SYSTEM DRILL_MVCDR (* Drill System Control+Diagnostics+HMI with Remote Model+View *)
  (* Standard: 61499-1; Classification: Simulation; ApplicationDomain: Transfer Lines; Function: Drilling *)
  (* Version 0.1, 2004-10-19, JHC, Rockwell Automation, Extended from DRILL_MVCDL. *)
  (* Version 0.0, 2004-09-28, JHC, Rockwell Automation, Extended from DRILL_MVCDL1. *)
  DEVICE MODEL : RMT_FRAME
    RESOURCE CLOCK : EMB_RES
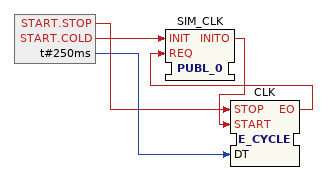
      FBS
        CLK : E_CYCLE;
        SIM_CLK : PUBL_0;
      END_FBS
      EVENT_CONNECTIONS
        START.STOP TO CLK.STOP;
        START.COLD TO SIM_CLK.INIT;
        SIM_CLK.INITO TO CLK.START;
        CLK.EO TO SIM_CLK.REQ;
      END_CONNECTIONS
      DATA_CONNECTIONS
        t#250ms TO CLK.DT;
      END_CONNECTIONS
    END_RESOURCE
    RESOURCE SENSORS : EMB_RES (* Sensor Data Concentrator/Publisher *)
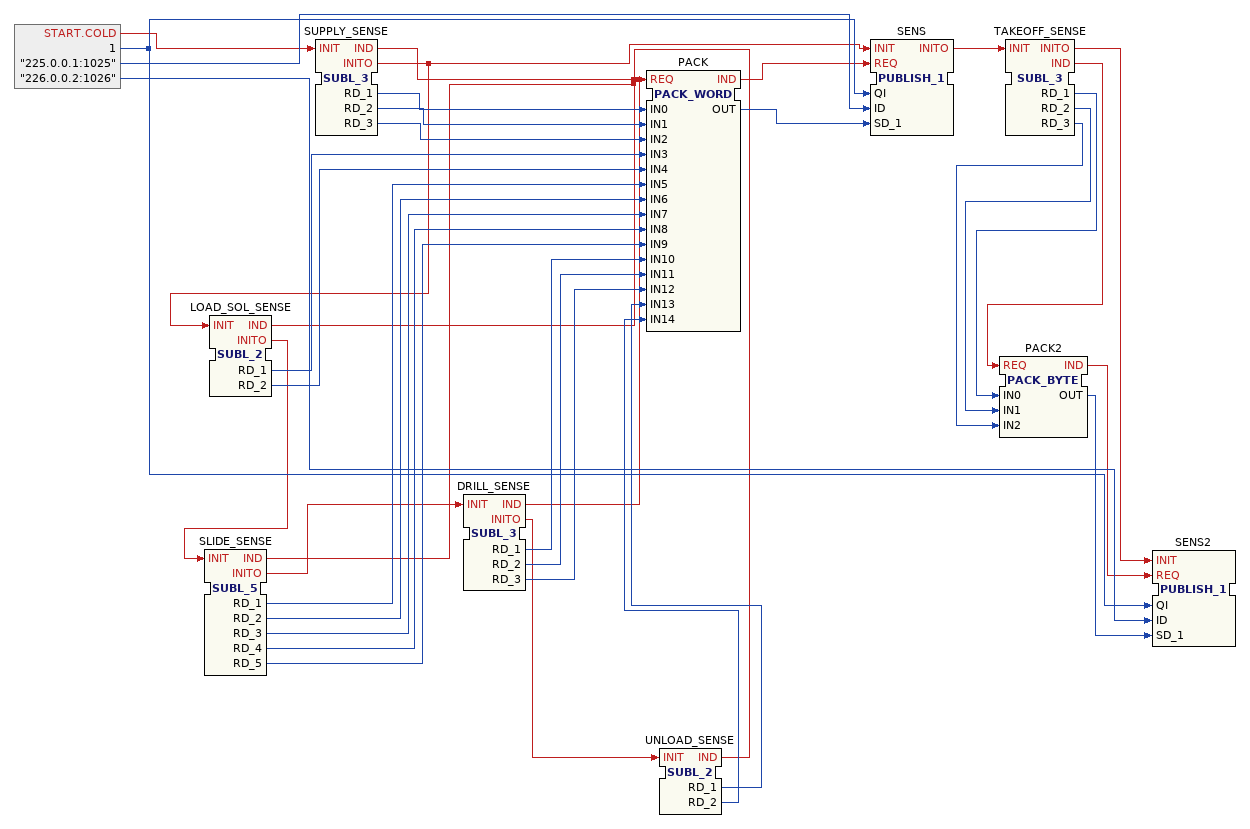
      FBS
        PACK : PACK_WORD;
        SENS : PUBLISH_1;
        SUPPLY_SENSE : SUBL_3;
        LOAD_SOL_SENSE : SUBL_2;
        SLIDE_SENSE : SUBL_5;
        DRILL_SENSE : SUBL_3;
        UNLOAD_SENSE : SUBL_2;
        SENS2 : PUBLISH_1;
        PACK2 : PACK_BYTE;
        TAKEOFF_SENSE : SUBL_3;
      END_FBS
      EVENT_CONNECTIONS
        SUPPLY_SENSE.IND TO PACK.REQ;
        LOAD_SOL_SENSE.IND TO PACK.REQ;
        SLIDE_SENSE.IND TO PACK.REQ;
        START.COLD TO SUPPLY_SENSE.INIT;
        DRILL_SENSE.IND TO PACK.REQ;
        SUPPLY_SENSE.INITO TO LOAD_SOL_SENSE.INIT;
        LOAD_SOL_SENSE.INITO TO SLIDE_SENSE.INIT;
        SLIDE_SENSE.INITO TO DRILL_SENSE.INIT;
        DRILL_SENSE.INITO TO UNLOAD_SENSE.INIT;
        UNLOAD_SENSE.IND TO PACK.REQ;
        SUPPLY_SENSE.INITO TO SENS.INIT;
        SENS.INITO TO TAKEOFF_SENSE.INIT;
        TAKEOFF_SENSE.INITO TO SENS2.INIT;
        PACK.IND TO SENS.REQ;
        TAKEOFF_SENSE.IND TO PACK2.REQ;
        PACK2.IND TO SENS2.REQ;
      END_CONNECTIONS
      DATA_CONNECTIONS
        SUPPLY_SENSE.RD_1 TO PACK.IN0;
        SUPPLY_SENSE.RD_2 TO PACK.IN1;
        SUPPLY_SENSE.RD_3 TO PACK.IN2;
        LOAD_SOL_SENSE.RD_1 TO PACK.IN3;
        LOAD_SOL_SENSE.RD_2 TO PACK.IN4;
        SLIDE_SENSE.RD_1 TO PACK.IN5;
        SLIDE_SENSE.RD_2 TO PACK.IN6;
        SLIDE_SENSE.RD_3 TO PACK.IN7;
        SLIDE_SENSE.RD_4 TO PACK.IN8;
        SLIDE_SENSE.RD_5 TO PACK.IN9;
        DRILL_SENSE.RD_1 TO PACK.IN10;
        DRILL_SENSE.RD_2 TO PACK.IN11;
        DRILL_SENSE.RD_3 TO PACK.IN12;
        UNLOAD_SENSE.RD_1 TO PACK.IN13;
        UNLOAD_SENSE.RD_2 TO PACK.IN14;
        1 TO SENS.QI;
        "225.0.0.1:1025" TO SENS.ID;
        PACK.OUT TO SENS.SD_1;
        TAKEOFF_SENSE.RD_1 TO PACK2.IN0;
        TAKEOFF_SENSE.RD_2 TO PACK2.IN1;
        TAKEOFF_SENSE.RD_3 TO PACK2.IN2;
        1 TO SENS2.QI;
        "226.0.0.2:1026" TO SENS2.ID;
        PACK2.OUT TO SENS2.SD_1;
      END_CONNECTIONS
    END_RESOURCE
    RESOURCE ACTUATORS : EMB_RES (* Actuator Data Subscriber/Distributor *)
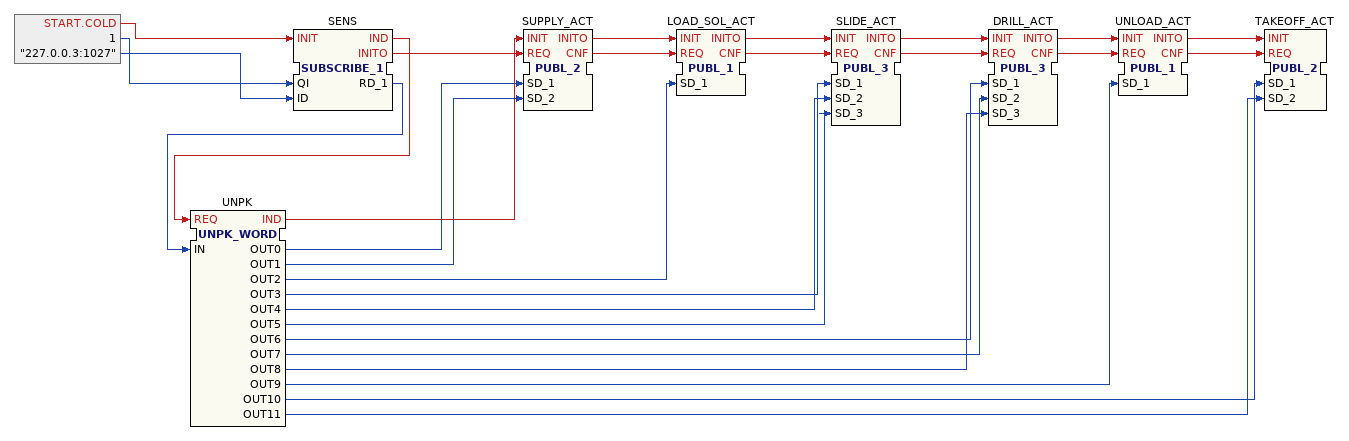
      FBS
        UNPK : UNPK_WORD;
        SENS : SUBSCRIBE_1;
        SUPPLY_ACT : PUBL_2;
        LOAD_SOL_ACT : PUBL_1;
        SLIDE_ACT : PUBL_3;
        DRILL_ACT : PUBL_3;
        UNLOAD_ACT : PUBL_1;
        TAKEOFF_ACT : PUBL_2;
      END_FBS
      EVENT_CONNECTIONS
        START.COLD TO SENS.INIT;
        SENS.IND TO UNPK.REQ;
        SENS.INITO TO SUPPLY_ACT.INIT;
        UNPK.IND TO SUPPLY_ACT.REQ;
        SUPPLY_ACT.INITO TO LOAD_SOL_ACT.INIT;
        SUPPLY_ACT.CNF TO LOAD_SOL_ACT.REQ;
        LOAD_SOL_ACT.INITO TO SLIDE_ACT.INIT;
        LOAD_SOL_ACT.CNF TO SLIDE_ACT.REQ;
        SLIDE_ACT.INITO TO DRILL_ACT.INIT;
        SLIDE_ACT.CNF TO DRILL_ACT.REQ;
        DRILL_ACT.INITO TO UNLOAD_ACT.INIT;
        DRILL_ACT.CNF TO UNLOAD_ACT.REQ;
        UNLOAD_ACT.INITO TO TAKEOFF_ACT.INIT;
        UNLOAD_ACT.CNF TO TAKEOFF_ACT.REQ;
      END_CONNECTIONS
      DATA_CONNECTIONS
        1 TO SENS.QI;
        "227.0.0.3:1027" TO SENS.ID;
        SENS.RD_1 TO UNPK.IN;
        UNPK.OUT0 TO SUPPLY_ACT.SD_1;
        UNPK.OUT1 TO SUPPLY_ACT.SD_2;
        UNPK.OUT2 TO LOAD_SOL_ACT.SD_1;
        UNPK.OUT3 TO SLIDE_ACT.SD_1;
        UNPK.OUT4 TO SLIDE_ACT.SD_2;
        UNPK.OUT5 TO SLIDE_ACT.SD_3;
        UNPK.OUT6 TO DRILL_ACT.SD_1;
        UNPK.OUT7 TO DRILL_ACT.SD_2;
        UNPK.OUT8 TO DRILL_ACT.SD_3;
        UNPK.OUT9 TO UNLOAD_ACT.SD_1;
        UNPK.OUT10 TO TAKEOFF_ACT.SD_1;
        UNPK.OUT11 TO TAKEOFF_ACT.SD_2;
      END_CONNECTIONS
    END_RESOURCE
    RESOURCE SUPPLY_MDL : EMB_RES
      FBS
        SUPPLY : XBAR_MDLL;
        LOAD_SOL : SOL_MDLL;
        UNLD : E_R_TRIG;
        LOAD : E_R_TRIG;
        SUPPLY_LOAD : LOADL;
      END_FBS
      EVENT_CONNECTIONS
        START.COLD TO SUPPLY.INIT;
        LOAD_SOL.IND TO UNLD.EI;
        SUPPLY.IND TO LOAD.EI;
        UNLD.EO TO SUPPLY.UNLD;
        SUPPLY.INITO TO SUPPLY_LOAD.INIT;
        SUPPLY_LOAD.INITO TO LOAD_SOL.INIT;
        LOAD_SOL.INITO TO SUPPLY_LOAD.REQ;
        LOAD.EO TO SUPPLY_LOAD.REQ;
      END_CONNECTIONS
      DATA_CONNECTIONS
        34 TO LOAD_SOL.VF;
        50 TO LOAD_SOL.VR;
        LOAD_SOL.END TO UNLD.QI;
        5 TO SUPPLY.VF;
        10 TO SUPPLY.VR;
        SUPPLY.HOME TO LOAD.QI;
        0 TO SUPPLY_LOAD.LPOS;
        VSTYLE#DISC TO SUPPLY_LOAD.STYLE;
        [255,255,0] TO SUPPLY_LOAD.WKPC;
      END_CONNECTIONS
    END_RESOURCE
    RESOURCE SLIDE_MDL : EMB_RES
      FBS
        SLIDE : XSLIDE_MDLL;
        UNLOAD : SOL_MDLL;
        DRILL_SENSE : SUBL_3;
        MAKE_HOLE : E_R_TRIG;
        UNLD : E_R_TRIG;
        LOAD_SOL_SENSE : SUBL_2;
        LOAD : E_R_TRIG;
        SLIDE_LOAD : LOADL;
        DRILLIT : LOADL;
      END_FBS
      EVENT_CONNECTIONS
        DRILL_SENSE.IND TO MAKE_HOLE.EI;
        UNLOAD.IND TO UNLD.EI;
        UNLD.EO TO SLIDE.UNLD;
        LOAD_SOL_SENSE.IND TO LOAD.EI;
        START.COLD TO UNLOAD.INIT;
        UNLOAD.INITO TO SLIDE.INIT;
        SLIDE.INITO TO LOAD_SOL_SENSE.INIT;
        LOAD_SOL_SENSE.INITO TO SLIDE_LOAD.INIT;
        LOAD.EO TO SLIDE_LOAD.REQ;
        MAKE_HOLE.EO TO DRILLIT.REQ;
        DRILLIT.INITO TO SLIDE.UNLD;
        SLIDE_LOAD.INITO TO DRILL_SENSE.INIT;
        DRILL_SENSE.INITO TO DRILLIT.INIT;
      END_CONNECTIONS
      DATA_CONNECTIONS
        50 TO UNLOAD.VF;
        50 TO UNLOAD.VR;
        DRILL_SENSE.RD_2 TO MAKE_HOLE.QI;
        20 TO SLIDE.VF;
        20 TO SLIDE.VR;
        UNLOAD.END TO UNLD.QI;
        LOAD_SOL_SENSE.RD_2 TO LOAD.QI;
        0 TO SLIDE_LOAD.LPOS;
        VSTYLE#DISC TO SLIDE_LOAD.STYLE;
        [255,255,0] TO SLIDE_LOAD.WKPC;
        "SLIDE_LOAD" TO DRILLIT.ID;
        100 TO DRILLIT.LPOS;
        VSTYLE#RING TO DRILLIT.STYLE;
        [255,255,0] TO DRILLIT.WKPC;
      END_CONNECTIONS
    END_RESOURCE
    RESOURCE DRILL_MDL : EMB_RES
      FBS
        DRILL : XBAR_MDLL;
        DRILL_ACT : SUBL_3;
        TOOL : E_SWITCH;
        DRILL_LOAD : LOADL;
        DRILL_UNLD : LOADL;
      END_FBS
      EVENT_CONNECTIONS
        START.COLD TO DRILL_ACT.INIT;
        DRILL_ACT.INITO TO DRILL.INIT;
        DRILL.INITO TO DRILL_LOAD.INIT;
        DRILL_LOAD.INITO TO DRILL_UNLD.INIT;
        DRILL_ACT.IND TO TOOL.EI;
        TOOL.EO1 TO DRILL_LOAD.REQ;
        TOOL.EO0 TO DRILL_UNLD.REQ;
        DRILL_UNLD.INITO TO DRILL_UNLD.REQ;
      END_CONNECTIONS
      DATA_CONNECTIONS
        10 TO DRILL.VF;
        15 TO DRILL.VR;
        VSTYLE#TOOL_ON TO DRILL_LOAD.STYLE;
        [255,255,0] TO DRILL_LOAD.WKPC;
        "DRILL_LOAD" TO DRILL_UNLD.ID;
        VSTYLE#TOOL_OFF TO DRILL_UNLD.STYLE;
        [255,255,0] TO DRILL_UNLD.WKPC;
        DRILL_ACT.RD_3 TO TOOL.G;
      END_CONNECTIONS
    END_RESOURCE
    RESOURCE TAKEOFF_MDL : EMB_RES
      FBS
        UNLOAD_SENSE : SUBL_2;
        TAKEOFF : XBAR_MDLL;
        UNLD : E_R_TRIG;
        LOAD : E_R_TRIG;
        TAKEOFF_LOAD : LOADL;
      END_FBS
      EVENT_CONNECTIONS
        START.COLD TO UNLOAD_SENSE.INIT;
        UNLD.EO TO TAKEOFF.UNLD;
        TAKEOFF.IND TO UNLD.EI;
        TAKEOFF.INITO TO TAKEOFF.UNLD;
        UNLOAD_SENSE.IND TO LOAD.EI;
        UNLOAD_SENSE.INITO TO TAKEOFF_LOAD.INIT;
        TAKEOFF_LOAD.INITO TO TAKEOFF.INIT;
        LOAD.EO TO TAKEOFF_LOAD.REQ;
      END_CONNECTIONS
      DATA_CONNECTIONS
        TAKEOFF.END TO UNLD.QI;
        10 TO TAKEOFF.VF;
        10 TO TAKEOFF.VR;
        UNLOAD_SENSE.RD_2 TO LOAD.QI;
        0 TO TAKEOFF_LOAD.LPOS;
        VSTYLE#RING TO TAKEOFF_LOAD.STYLE;
        [255,255,0] TO TAKEOFF_LOAD.WKPC;
      END_CONNECTIONS
    END_RESOURCE
    RESOURCE INPUT_VIEW : VIEW_PANEL
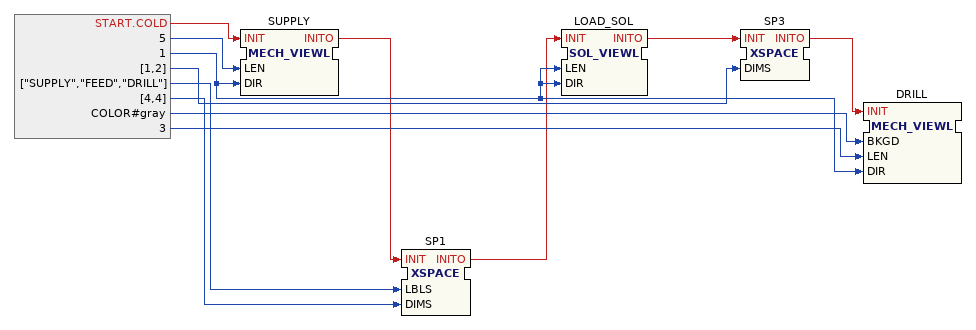
      FBS
        SUPPLY : MECH_VIEWL; (* Supply transfer mechanism *)
        SP1 : XSPACE;
        LOAD_SOL : SOL_VIEWL; (* Loader mechanism *)
        SP3 : XSPACE;
        DRILL : MECH_VIEWL;
      END_FBS
      EVENT_CONNECTIONS
        START.COLD TO SUPPLY.INIT;
        SUPPLY.INITO TO SP1.INIT;
        SP1.INITO TO LOAD_SOL.INIT;
        LOAD_SOL.INITO TO SP3.INIT;
        SP3.INITO TO DRILL.INIT;
      END_CONNECTIONS
      DATA_CONNECTIONS
        5 TO SUPPLY.LEN;
        1 TO SUPPLY.DIR;
        [1,2] TO SP3.DIMS;
        ["SUPPLY","FEED","DRILL"] TO SP1.LBLS;
        [4,4] TO SP1.DIMS;
        COLOR#gray TO DRILL.BKGD;
        3 TO DRILL.LEN;
        1 TO DRILL.DIR;
        1 TO LOAD_SOL.LEN;
        1 TO LOAD_SOL.DIR;
      END_CONNECTIONS
    END_RESOURCE
    RESOURCE OUTPUT_VIEW : VIEW_PANEL
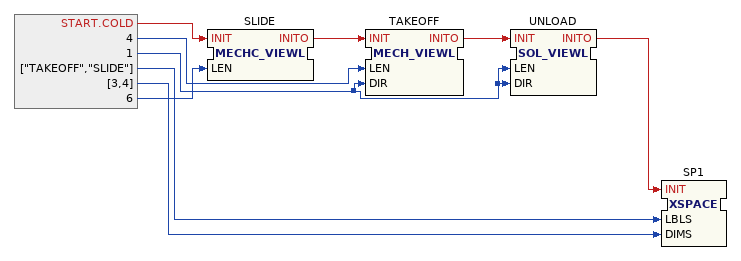
      FBS
        SLIDE : MECHC_VIEWL;
        TAKEOFF : MECH_VIEWL; (* Takeoff Transfer *)
        UNLOAD : SOL_VIEWL; (* Unloader Mechanism *)
        SP1 : XSPACE;
      END_FBS
      EVENT_CONNECTIONS
        START.COLD TO SLIDE.INIT;
        SLIDE.INITO TO TAKEOFF.INIT;
        TAKEOFF.INITO TO UNLOAD.INIT;
        UNLOAD.INITO TO SP1.INIT;
      END_CONNECTIONS
      DATA_CONNECTIONS
        4 TO TAKEOFF.LEN;
        1 TO TAKEOFF.DIR;
        ["TAKEOFF","SLIDE"] TO SP1.LBLS;
        [3,4] TO SP1.DIMS;
        1 TO UNLOAD.LEN;
        1 TO UNLOAD.DIR;
        6 TO SLIDE.LEN;
      END_CONNECTIONS
    END_RESOURCE
    DATA_CONNECTIONS
      0 TO INPUT_VIEW.TRACE;
      30 TO INPUT_VIEW.DIA;
      [6,5] TO INPUT_VIEW.SIZE;
      1 TO INPUT_VIEW.VERTICAL;
      30 TO OUTPUT_VIEW.DIA;
      [6,5] TO OUTPUT_VIEW.SIZE;
    END_CONNECTIONS
  END_DEVICE
  DEVICE DIAGNOSTICS : FRAME_DEVICE
    RESOURCE LOG : PANEL_RESOURCE
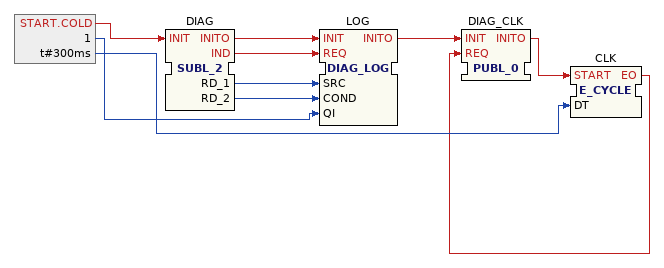
      FBS
        DIAG : SUBL_2;
        LOG : DIAG_LOG;
        CLK : E_CYCLE;
        DIAG_CLK : PUBL_0;
      END_FBS
      EVENT_CONNECTIONS
        START.COLD TO DIAG.INIT;
        DIAG.INITO TO LOG.INIT;
        DIAG.IND TO LOG.REQ;
        LOG.INITO TO DIAG_CLK.INIT;
        DIAG_CLK.INITO TO CLK.START;
        CLK.EO TO DIAG_CLK.REQ;
      END_CONNECTIONS
      DATA_CONNECTIONS
        DIAG.RD_1 TO LOG.SRC;
        DIAG.RD_2 TO LOG.COND;
        1 TO LOG.QI;
        t#300ms TO CLK.DT; (* Stretched 20% from MODEL.CLOCK.CLK.DT *)
      END_CONNECTIONS
    END_RESOURCE
    RESOURCE MONITOR : EMB_RES
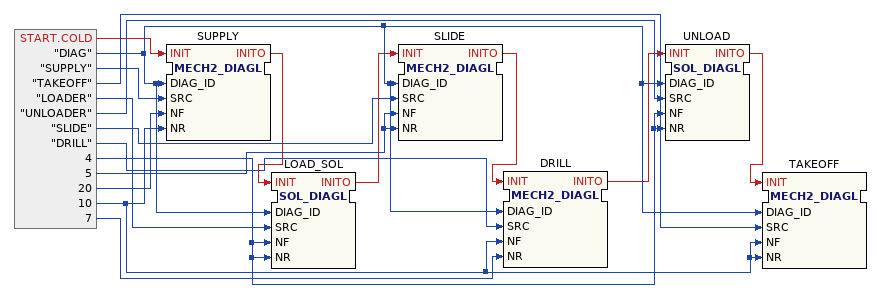
      FBS
        SUPPLY : MECH2_DIAGL;
        LOAD_SOL : SOL_DIAGL;
        SLIDE : MECH2_DIAGL;
        DRILL : MECH2_DIAGL;
        UNLOAD : SOL_DIAGL;
        TAKEOFF : MECH2_DIAGL;
      END_FBS
      EVENT_CONNECTIONS
        START.COLD TO SUPPLY.INIT;
        SUPPLY.INITO TO LOAD_SOL.INIT;
        LOAD_SOL.INITO TO SLIDE.INIT;
        SLIDE.INITO TO DRILL.INIT;
        DRILL.INITO TO UNLOAD.INIT;
        UNLOAD.INITO TO TAKEOFF.INIT;
      END_CONNECTIONS
      DATA_CONNECTIONS
        "DIAG" TO SUPPLY.DIAG_ID;
        "SUPPLY" TO SUPPLY.SRC;
        "DIAG" TO TAKEOFF.DIAG_ID;
        "TAKEOFF" TO TAKEOFF.SRC;
        "DIAG" TO LOAD_SOL.DIAG_ID;
        "LOADER" TO LOAD_SOL.SRC;
        "DIAG" TO UNLOAD.DIAG_ID;
        "UNLOADER" TO UNLOAD.SRC;
        "DIAG" TO SLIDE.DIAG_ID;
        "SLIDE" TO SLIDE.SRC;
        "DIAG" TO DRILL.DIAG_ID;
        "DRILL" TO DRILL.SRC;
        4 TO UNLOAD.NF;
        4 TO UNLOAD.NR;
        4 TO LOAD_SOL.NF;
        4 TO LOAD_SOL.NR;
        5 TO SLIDE.NF;
        5 TO SLIDE.NR;
        20 TO SUPPLY.NF;
        10 TO SUPPLY.NR;
        10 TO TAKEOFF.NF;
        10 TO TAKEOFF.NR;
        10 TO DRILL.NF;
        7 TO DRILL.NR;
      END_CONNECTIONS
    END_RESOURCE
    RESOURCE CLAMP : EMB_RES (* Special Monitoring for Clamp *)
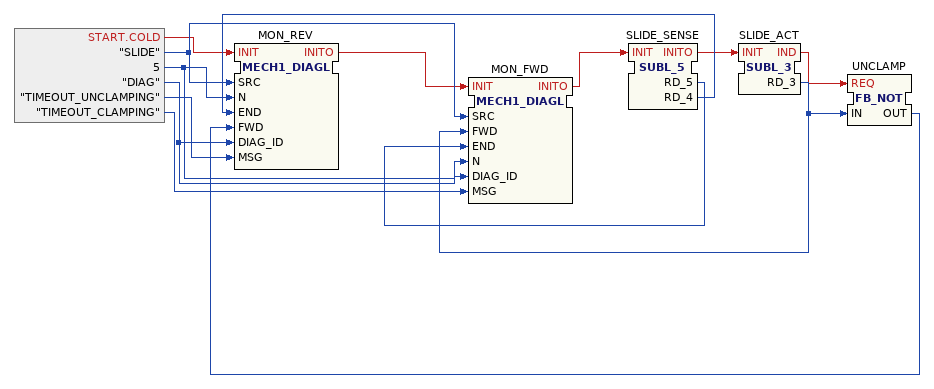
      FBS
        MON_FWD : MECH1_DIAGL;
        SLIDE_ACT : SUBL_3;
        SLIDE_SENSE : SUBL_5;
        MON_REV : MECH1_DIAGL;
        UNCLAMP : FB_NOT;
      END_FBS
      EVENT_CONNECTIONS
        SLIDE_ACT.IND TO UNCLAMP.REQ;
        SLIDE_SENSE.INITO TO SLIDE_ACT.INIT;
        START.COLD TO MON_REV.INIT;
        MON_REV.INITO TO MON_FWD.INIT;
        MON_FWD.INITO TO SLIDE_SENSE.INIT;
      END_CONNECTIONS
      DATA_CONNECTIONS
        "SLIDE" TO MON_FWD.SRC;
        "SLIDE" TO MON_REV.SRC;
        SLIDE_ACT.RD_3 TO UNCLAMP.IN;
        SLIDE_ACT.RD_3 TO MON_FWD.FWD;
        SLIDE_SENSE.RD_5 TO MON_FWD.END;
        5 TO MON_FWD.N;
        5 TO MON_REV.N;
        SLIDE_SENSE.RD_4 TO MON_REV.END;
        UNCLAMP.OUT TO MON_REV.FWD;
        "DIAG" TO MON_FWD.DIAG_ID;
        "DIAG" TO MON_REV.DIAG_ID;
        "TIMEOUT_UNCLAMPING" TO MON_REV.MSG;
        "TIMEOUT_CLAMPING" TO MON_FWD.MSG;
      END_CONNECTIONS
    END_RESOURCE
    RESOURCE SENSORS : EMB_RES (* Subscriber/Distributor for Sensors *)
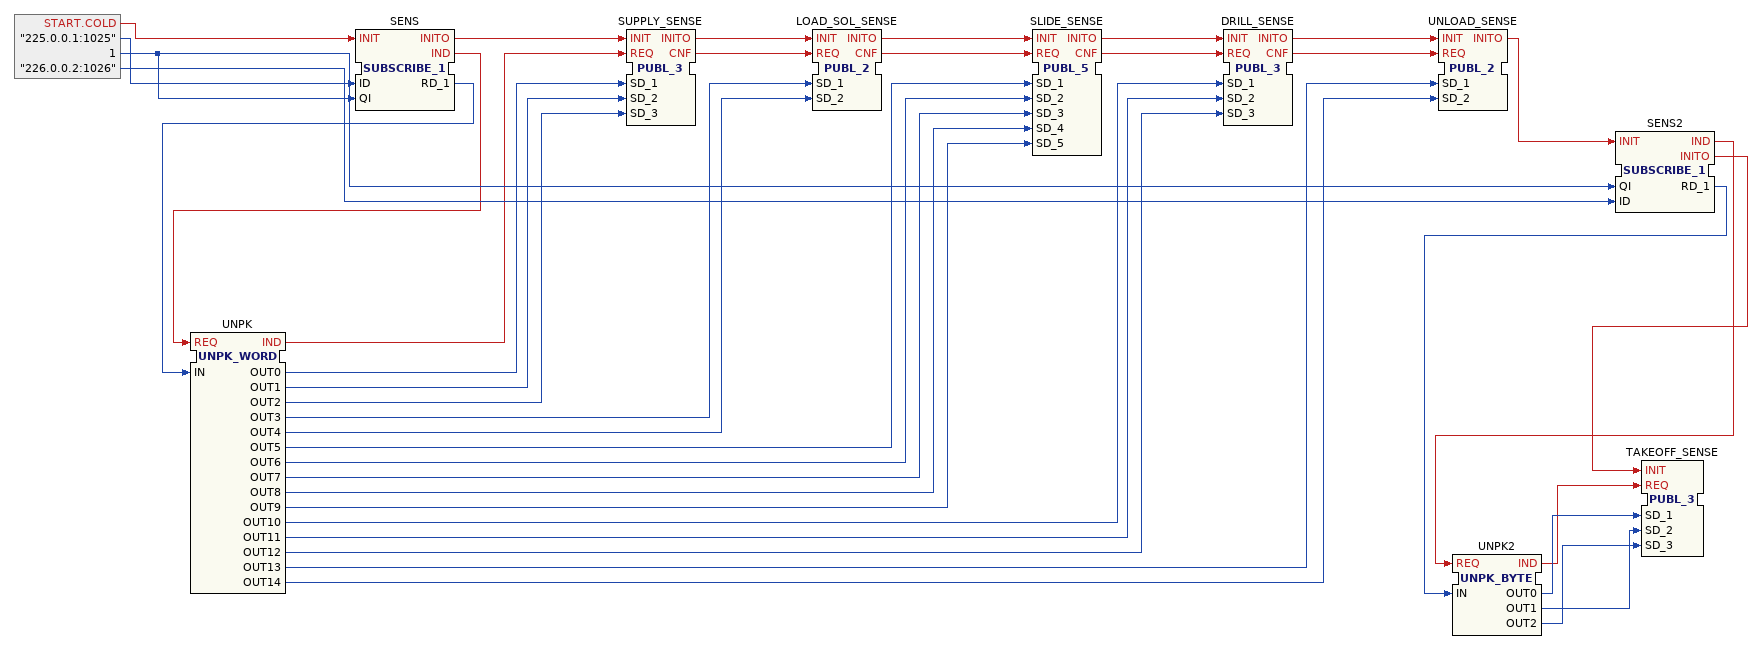
      FBS
        UNPK : UNPK_WORD;
        SENS : SUBSCRIBE_1;
        SUPPLY_SENSE : PUBL_3;
        LOAD_SOL_SENSE : PUBL_2;
        SLIDE_SENSE : PUBL_5;
        DRILL_SENSE : PUBL_3;
        UNLOAD_SENSE : PUBL_2;
        SENS2 : SUBSCRIBE_1;
        UNPK2 : UNPK_BYTE;
        TAKEOFF_SENSE : PUBL_3;
      END_FBS
      EVENT_CONNECTIONS
        START.COLD TO SENS.INIT;
        SENS.INITO TO SUPPLY_SENSE.INIT;
        SENS.IND TO UNPK.REQ;
        UNPK.IND TO SUPPLY_SENSE.REQ;
        SUPPLY_SENSE.INITO TO LOAD_SOL_SENSE.INIT;
        SUPPLY_SENSE.CNF TO LOAD_SOL_SENSE.REQ;
        LOAD_SOL_SENSE.INITO TO SLIDE_SENSE.INIT;
        LOAD_SOL_SENSE.CNF TO SLIDE_SENSE.REQ;
        SLIDE_SENSE.INITO TO DRILL_SENSE.INIT;
        SLIDE_SENSE.CNF TO DRILL_SENSE.REQ;
        DRILL_SENSE.INITO TO UNLOAD_SENSE.INIT;
        DRILL_SENSE.CNF TO UNLOAD_SENSE.REQ;
        UNLOAD_SENSE.INITO TO SENS2.INIT;
        SENS2.IND TO UNPK2.REQ;
        SENS2.INITO TO TAKEOFF_SENSE.INIT;
        UNPK2.IND TO TAKEOFF_SENSE.REQ;
      END_CONNECTIONS
      DATA_CONNECTIONS
        UNPK.OUT0 TO SUPPLY_SENSE.SD_1;
        UNPK.OUT1 TO SUPPLY_SENSE.SD_2;
        UNPK.OUT2 TO SUPPLY_SENSE.SD_3;
        UNPK.OUT3 TO LOAD_SOL_SENSE.SD_1;
        UNPK.OUT4 TO LOAD_SOL_SENSE.SD_2;
        SENS.RD_1 TO UNPK.IN;
        UNPK.OUT5 TO SLIDE_SENSE.SD_1;
        UNPK.OUT6 TO SLIDE_SENSE.SD_2;
        UNPK.OUT7 TO SLIDE_SENSE.SD_3;
        UNPK.OUT8 TO SLIDE_SENSE.SD_4;
        UNPK.OUT9 TO SLIDE_SENSE.SD_5;
        UNPK.OUT10 TO DRILL_SENSE.SD_1;
        UNPK.OUT11 TO DRILL_SENSE.SD_2;
        UNPK.OUT12 TO DRILL_SENSE.SD_3;
        "225.0.0.1:1025" TO SENS.ID;
        UNPK.OUT13 TO UNLOAD_SENSE.SD_1;
        UNPK.OUT14 TO UNLOAD_SENSE.SD_2;
        1 TO SENS2.QI;
        1 TO SENS.QI;
        SENS2.RD_1 TO UNPK2.IN;
        UNPK2.OUT0 TO TAKEOFF_SENSE.SD_1;
        UNPK2.OUT1 TO TAKEOFF_SENSE.SD_2;
        "226.0.0.2:1026" TO SENS2.ID;
        UNPK2.OUT2 TO TAKEOFF_SENSE.SD_3;
      END_CONNECTIONS
    END_RESOURCE
    RESOURCE ACTUATORS : EMB_RES (* Collector/Publisher for Actuators *)
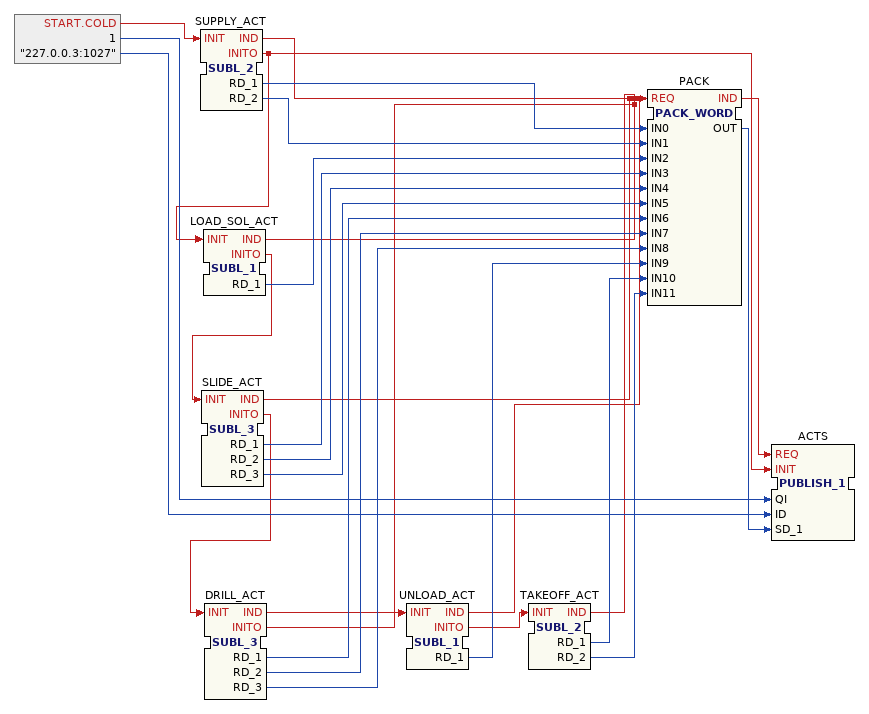
      FBS
        PACK : PACK_WORD;
        ACTS : PUBLISH_1;
        SUPPLY_ACT : SUBL_2;
        LOAD_SOL_ACT : SUBL_1;
        SLIDE_ACT : SUBL_3;
        DRILL_ACT : SUBL_3;
        UNLOAD_ACT : SUBL_1;
        TAKEOFF_ACT : SUBL_2;
      END_FBS
      EVENT_CONNECTIONS
        PACK.IND TO ACTS.REQ;
        SUPPLY_ACT.IND TO PACK.REQ;
        LOAD_SOL_ACT.IND TO PACK.REQ;
        SLIDE_ACT.IND TO PACK.REQ;
        DRILL_ACT.IND TO PACK.REQ;
        UNLOAD_ACT.IND TO PACK.REQ;
        TAKEOFF_ACT.IND TO PACK.REQ;
        START.COLD TO SUPPLY_ACT.INIT;
        SUPPLY_ACT.INITO TO LOAD_SOL_ACT.INIT;
        LOAD_SOL_ACT.INITO TO SLIDE_ACT.INIT;
        SLIDE_ACT.INITO TO DRILL_ACT.INIT;
        DRILL_ACT.INITO TO UNLOAD_ACT.INIT;
        UNLOAD_ACT.INITO TO TAKEOFF_ACT.INIT;
        SUPPLY_ACT.INITO TO ACTS.INIT;
      END_CONNECTIONS
      DATA_CONNECTIONS
        1 TO ACTS.QI;
        "227.0.0.3:1027" TO ACTS.ID;
        PACK.OUT TO ACTS.SD_1;
        SUPPLY_ACT.RD_1 TO PACK.IN0;
        SUPPLY_ACT.RD_2 TO PACK.IN1;
        LOAD_SOL_ACT.RD_1 TO PACK.IN2;
        SLIDE_ACT.RD_1 TO PACK.IN3;
        SLIDE_ACT.RD_2 TO PACK.IN4;
        SLIDE_ACT.RD_3 TO PACK.IN5;
        DRILL_ACT.RD_1 TO PACK.IN6;
        DRILL_ACT.RD_2 TO PACK.IN7;
        DRILL_ACT.RD_3 TO PACK.IN8;
        UNLOAD_ACT.RD_1 TO PACK.IN9;
        TAKEOFF_ACT.RD_1 TO PACK.IN10;
        TAKEOFF_ACT.RD_2 TO PACK.IN11;
      END_CONNECTIONS
    END_RESOURCE
    DATA_CONNECTIONS
      1 TO LOG.ROWS;
      1 TO LOG.COLS;
    END_CONNECTIONS
  END_DEVICE
  DEVICE CONTROL : FRAME_DEVICE
    RESOURCE SUPPLY_SENSORS : PANEL_RESOURCE
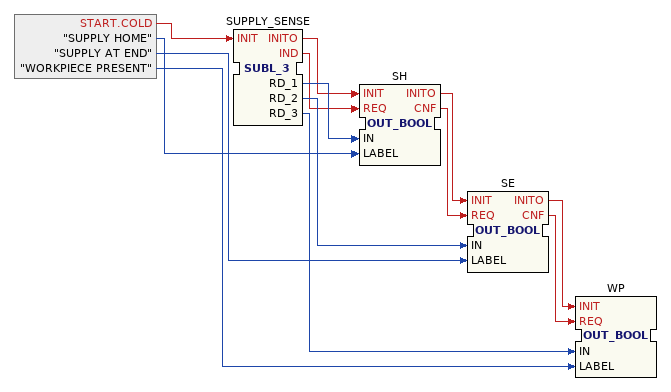
      FBS
        SUPPLY_SENSE : SUBL_3;
        SH : OUT_BOOL;
        SE : OUT_BOOL;
        WP : OUT_BOOL;
      END_FBS
      EVENT_CONNECTIONS
        START.COLD TO SUPPLY_SENSE.INIT;
        SUPPLY_SENSE.INITO TO SH.INIT;
        SH.INITO TO SE.INIT;
        SE.INITO TO WP.INIT;
        SUPPLY_SENSE.IND TO SH.REQ;
        SH.CNF TO SE.REQ;
        SE.CNF TO WP.REQ;
      END_CONNECTIONS
      DATA_CONNECTIONS
        SUPPLY_SENSE.RD_1 TO SH.IN;
        SUPPLY_SENSE.RD_2 TO SE.IN;
        SUPPLY_SENSE.RD_3 TO WP.IN;
        "SUPPLY HOME" TO SH.LABEL;
        "SUPPLY AT END" TO SE.LABEL;
        "WORKPIECE PRESENT" TO WP.LABEL;
      END_CONNECTIONS
    END_RESOURCE
    RESOURCE SUPPLY_ACTUATORS : PANEL_RESOURCE
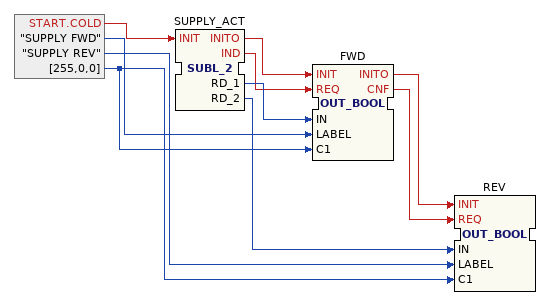
      FBS
        FWD : OUT_BOOL;
        REV : OUT_BOOL;
        SUPPLY_ACT : SUBL_2;
      END_FBS
      EVENT_CONNECTIONS
        FWD.INITO TO REV.INIT;
        START.COLD TO SUPPLY_ACT.INIT;
        SUPPLY_ACT.INITO TO FWD.INIT;
        SUPPLY_ACT.IND TO FWD.REQ;
        FWD.CNF TO REV.REQ;
      END_CONNECTIONS
      DATA_CONNECTIONS
        SUPPLY_ACT.RD_1 TO FWD.IN;
        SUPPLY_ACT.RD_2 TO REV.IN;
        "SUPPLY FWD" TO FWD.LABEL;
        "SUPPLY REV" TO REV.LABEL;
        [255,0,0] TO FWD.C1;
        [255,0,0] TO REV.C1;
      END_CONNECTIONS
    END_RESOURCE
    RESOURCE LOAD_SENSORS : PANEL_RESOURCE
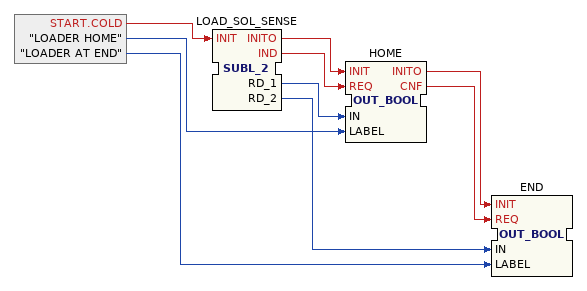
      FBS
        LOAD_SOL_SENSE : SUBL_2;
        HOME : OUT_BOOL;
        END : OUT_BOOL;
      END_FBS
      EVENT_CONNECTIONS
        START.COLD TO LOAD_SOL_SENSE.INIT;
        LOAD_SOL_SENSE.INITO TO HOME.INIT;
        HOME.INITO TO END.INIT;
        LOAD_SOL_SENSE.IND TO HOME.REQ;
        HOME.CNF TO END.REQ;
      END_CONNECTIONS
      DATA_CONNECTIONS
        LOAD_SOL_SENSE.RD_1 TO HOME.IN;
        LOAD_SOL_SENSE.RD_2 TO END.IN;
        "LOADER HOME" TO HOME.LABEL;
        "LOADER AT END" TO END.LABEL;
      END_CONNECTIONS
    END_RESOURCE
    RESOURCE LOAD_ACTUATORS : PANEL_RESOURCE
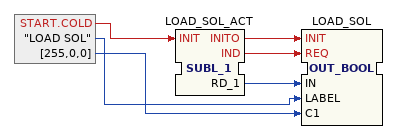
      FBS
        LOAD_SOL : OUT_BOOL;
        LOAD_SOL_ACT : SUBL_1;
      END_FBS
      EVENT_CONNECTIONS
        START.COLD TO LOAD_SOL_ACT.INIT;
        LOAD_SOL_ACT.INITO TO LOAD_SOL.INIT;
        LOAD_SOL_ACT.IND TO LOAD_SOL.REQ;
      END_CONNECTIONS
      DATA_CONNECTIONS
        LOAD_SOL_ACT.RD_1 TO LOAD_SOL.IN;
        "LOAD SOL" TO LOAD_SOL.LABEL;
        [255,0,0] TO LOAD_SOL.C1;
      END_CONNECTIONS
    END_RESOURCE
    RESOURCE SLIDE_SENSORS : PANEL_RESOURCE
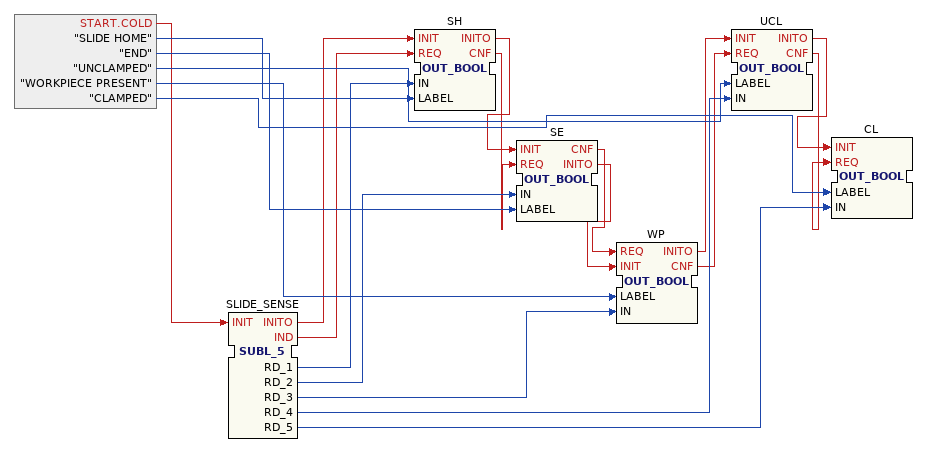
      FBS
        SLIDE_SENSE : SUBL_5;
        SH : OUT_BOOL;
        SE : OUT_BOOL;
        UCL : OUT_BOOL;
        CL : OUT_BOOL;
        WP : OUT_BOOL;
      END_FBS
      EVENT_CONNECTIONS
        START.COLD TO SLIDE_SENSE.INIT;
        SLIDE_SENSE.INITO TO SH.INIT;
        SH.INITO TO SE.INIT;
        UCL.INITO TO CL.INIT;
        SLIDE_SENSE.IND TO SH.REQ;
        SH.CNF TO SE.REQ;
        UCL.CNF TO CL.REQ;
        SE.CNF TO WP.REQ;
        SE.INITO TO WP.INIT;
        WP.INITO TO UCL.INIT;
        WP.CNF TO UCL.REQ;
      END_CONNECTIONS
      DATA_CONNECTIONS
        SLIDE_SENSE.RD_1 TO SH.IN;
        SLIDE_SENSE.RD_2 TO SE.IN;
        "SLIDE HOME" TO SH.LABEL;
        "END" TO SE.LABEL;
        "UNCLAMPED" TO UCL.LABEL;
        "WORKPIECE PRESENT" TO WP.LABEL;
        "CLAMPED" TO CL.LABEL;
        SLIDE_SENSE.RD_3 TO WP.IN;
        SLIDE_SENSE.RD_4 TO UCL.IN;
        SLIDE_SENSE.RD_5 TO CL.IN;
      END_CONNECTIONS
    END_RESOURCE
    RESOURCE SLIDE_ACTUATORS : PANEL_RESOURCE
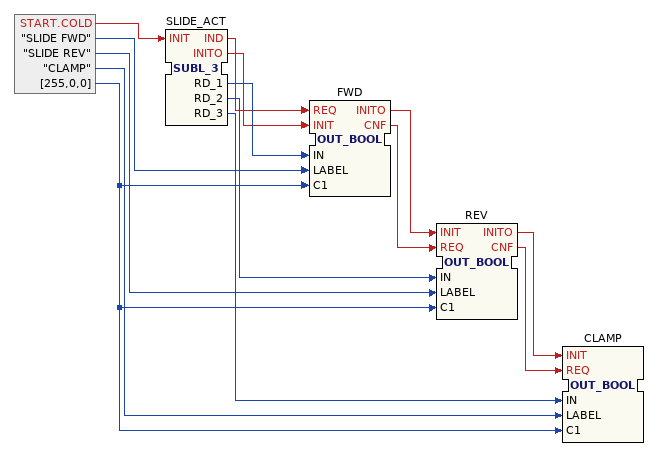
      FBS
        FWD : OUT_BOOL;
        REV : OUT_BOOL;
        CLAMP : OUT_BOOL;
        SLIDE_ACT : SUBL_3;
      END_FBS
      EVENT_CONNECTIONS
        FWD.INITO TO REV.INIT;
        REV.INITO TO CLAMP.INIT;
        REV.CNF TO CLAMP.REQ;
        FWD.CNF TO REV.REQ;
        START.COLD TO SLIDE_ACT.INIT;
        SLIDE_ACT.IND TO FWD.REQ;
        SLIDE_ACT.INITO TO FWD.INIT;
      END_CONNECTIONS
      DATA_CONNECTIONS
        SLIDE_ACT.RD_1 TO FWD.IN;
        SLIDE_ACT.RD_2 TO REV.IN;
        SLIDE_ACT.RD_3 TO CLAMP.IN;
        "SLIDE FWD" TO FWD.LABEL;
        "SLIDE REV" TO REV.LABEL;
        "CLAMP" TO CLAMP.LABEL;
        [255,0,0] TO FWD.C1;
        [255,0,0] TO REV.C1;
        [255,0,0] TO CLAMP.C1;
      END_CONNECTIONS
    END_RESOURCE
    RESOURCE DRILL_SENSORS : PANEL_RESOURCE
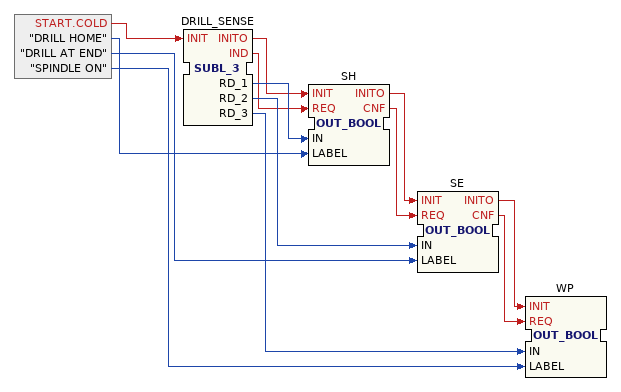
      FBS
        DRILL_SENSE : SUBL_3;
        SH : OUT_BOOL;
        SE : OUT_BOOL;
        WP : OUT_BOOL;
      END_FBS
      EVENT_CONNECTIONS
        START.COLD TO DRILL_SENSE.INIT;
        DRILL_SENSE.INITO TO SH.INIT;
        SH.INITO TO SE.INIT;
        SE.INITO TO WP.INIT;
        DRILL_SENSE.IND TO SH.REQ;
        SH.CNF TO SE.REQ;
        SE.CNF TO WP.REQ;
      END_CONNECTIONS
      DATA_CONNECTIONS
        DRILL_SENSE.RD_1 TO SH.IN;
        DRILL_SENSE.RD_2 TO SE.IN;
        DRILL_SENSE.RD_3 TO WP.IN;
        "DRILL HOME" TO SH.LABEL;
        "DRILL AT END" TO SE.LABEL;
        "SPINDLE ON" TO WP.LABEL;
      END_CONNECTIONS
    END_RESOURCE
    RESOURCE DRILL_ACTUATORS : PANEL_RESOURCE
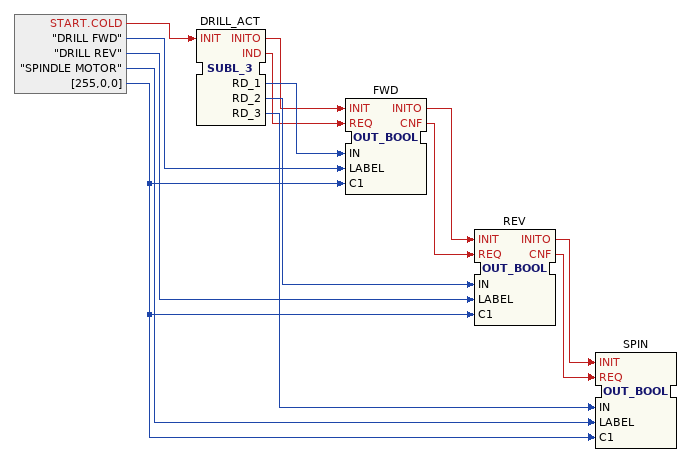
      FBS
        FWD : OUT_BOOL;
        REV : OUT_BOOL;
        SPIN : OUT_BOOL;
        DRILL_ACT : SUBL_3;
      END_FBS
      EVENT_CONNECTIONS
        FWD.INITO TO REV.INIT;
        REV.INITO TO SPIN.INIT;
        REV.CNF TO SPIN.REQ;
        FWD.CNF TO REV.REQ;
        START.COLD TO DRILL_ACT.INIT;
        DRILL_ACT.INITO TO FWD.INIT;
        DRILL_ACT.IND TO FWD.REQ;
      END_CONNECTIONS
      DATA_CONNECTIONS
        DRILL_ACT.RD_1 TO FWD.IN;
        DRILL_ACT.RD_2 TO REV.IN;
        DRILL_ACT.RD_3 TO SPIN.IN;
        "DRILL FWD" TO FWD.LABEL;
        "DRILL REV" TO REV.LABEL;
        "SPINDLE MOTOR" TO SPIN.LABEL;
        [255,0,0] TO FWD.C1;
        [255,0,0] TO REV.C1;
        [255,0,0] TO SPIN.C1;
      END_CONNECTIONS
    END_RESOURCE
    RESOURCE UNLOAD_SENSORS : PANEL_RESOURCE
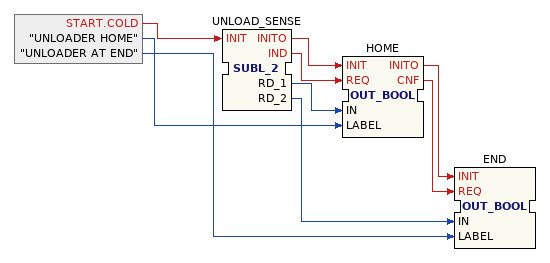
      FBS
        UNLOAD_SENSE : SUBL_2;
        HOME : OUT_BOOL;
        END : OUT_BOOL;
      END_FBS
      EVENT_CONNECTIONS
        START.COLD TO UNLOAD_SENSE.INIT;
        UNLOAD_SENSE.INITO TO HOME.INIT;
        HOME.INITO TO END.INIT;
        UNLOAD_SENSE.IND TO HOME.REQ;
        HOME.CNF TO END.REQ;
      END_CONNECTIONS
      DATA_CONNECTIONS
        UNLOAD_SENSE.RD_1 TO HOME.IN;
        UNLOAD_SENSE.RD_2 TO END.IN;
        "UNLOADER HOME" TO HOME.LABEL;
        "UNLOADER AT END" TO END.LABEL;
      END_CONNECTIONS
    END_RESOURCE
    RESOURCE UNLOAD_ACTUATORS : PANEL_RESOURCE
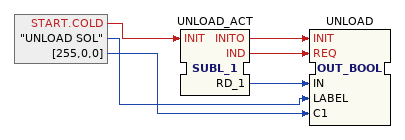
      FBS
        UNLOAD : OUT_BOOL;
        UNLOAD_ACT : SUBL_1;
      END_FBS
      EVENT_CONNECTIONS
        START.COLD TO UNLOAD_ACT.INIT;
        UNLOAD_ACT.INITO TO UNLOAD.INIT;
        UNLOAD_ACT.IND TO UNLOAD.REQ;
      END_CONNECTIONS
      DATA_CONNECTIONS
        UNLOAD_ACT.RD_1 TO UNLOAD.IN;
        "UNLOAD SOL" TO UNLOAD.LABEL;
        [255,0,0] TO UNLOAD.C1;
      END_CONNECTIONS
    END_RESOURCE
    RESOURCE TAKEOFF_SENSORS : PANEL_RESOURCE
